(* 
:Description: This function block is base for all other measurement fixtures.
*)
FUNCTION_BLOCK ABSTRACT FB_UniversalFixture IMPLEMENTS  I_UniversalFixture
VAR CONSTANT
	sSAMPLE_ACCEPTED : STRING := 'ACCEPTED';					(* Sample accepted - compare keyword for TCP/IP message from measurement device *)
	sSAMPLE_REJECTED : STRING := 'REJECTED';					(* Sample rejected - compare keyword for TCP/IP message from measurement device *)
END_VAR
VAR
	bFirstCycle				: BOOL := TRUE;						(* First cycle bit *)
	sName 					: STRING; 							(* Fixture name for other utilities *)
	
	bActive 				: BOOL;								(* Fixture device is initialized and ready to wokr *)
	bBusy					: BOOL;								(* Fixture device is busy *)
	bError 					: BOOL;								(* Error occured while executing *)
	iErrorID 				: UDINT;							(* Error ID *)
	
	eSampleResult			: E_UniversalFixtureSampleResult;	(* Result of current measured product *)
	iSampleID				: UDINT;							(* Id of current measured product *)
	bSocketOpen				: BOOL;								(* Socket open flag *)
	
	sSendData				: STRING;							(* String message to send via TCP/IP to measurement device *)
	sRecivedData			: STRING;							(* String message to recive via TCP/IP from measurement device *)
	sLoggerMessage			: STRING;							(* String message for measurement txt logger *)
	stSendData				: ST_TcpBufferData;					(* Byte message to send via TCP/IP to measurement device *)
	stReciveData			: ST_TcpBufferData;					(* Byte message to recive via TCP/IP from measurement device *)
	fbTcpServer				: FB_TcpServer;						(* TCP/IP server instance *)
	fbTcpClient				: FB_TcpClient;						(* TCP/IP client instance *)
	bUseLogger				: BOOL;								(* Enables using of internal fixture file logger *)
	fbMeasurementLogger 	: FB_TXTDataExchanger;				(* Measurement TXT-File logger *)
	
	rtError					: R_TRIG; 							(* Rising edge trigger for function block error *)
	
	eFixtureState			: E_UniversalFixtureState;			(* Current state of measurement fixture device *)
	eFixtureStateInit		: E_UniversalFixtureStateInit;		(* Current state of measurement fixture device initialization *)
	eFixtureStateAbort		: E_UniversalFixtureStateAbort;		(* Current state of measurement fixture device aborting *)
	eFixtureStateReset		: E_UniversalFixtureStateReset;		(* Current state of measurement fixture device reseting *)
	eFixtureStateMeasure	: E_UniversalFixtureStateMeasure; 	(* Current measurement state if measurement has began *)
	eConnnectionType		: E_UniversalFixtureConnectionType;
	
	bClientConnection 		: BOOL; 							(* If true then fixture connect as a client, if false it behaves like a server *)
END_VAR

(* First cycle assignamnets *)
IF bFirstCycle THEN
	bFirstCycle := FALSE;
	
END_IF

(* Update status flags *)
bActive := eFixtureState >= UNIVERSAL_FIXTURE_READY;
bError := fbTcpServer.Error OR fbMeasurementLogger.Error;

(* Run server instance *)
IF eConnnectionType = UNIVERSAL_FIXTURE_SERVER_CONNECTION THEN
	fbTcpServer();
	
ELSIF eConnnectionType = UNIVERSAL_FIXTURE_CLIENT_CONNECTION THEN
	fbTcpClient();
	
END_IF 

(* Report errors that occur *)
rtError(CLK:=bError);

IF rtError.Q THEN 
	fbMachineLogger.MR_AddLogs(FUN_MergeStrings5(sName, ' : Error occured (error ID: ', UDINT_TO_STRING(iErrorID), ')', ''));
	
END_IF

(* Run internal measurement logger instance if it's enabled *)
IF bUseLogger THEN
	fbMeasurementLogger();
	
END_IF

(* Run main state machine *)
StateMachine();

PROPERTY Active : REFERENCE TO BOOL
GET
Active REF= bActive;
END_GET
END_PROPERTY

PROPERTY Busy : REFERENCE TO BOOL
GET
Busy REF= bBusy;
END_GET
END_PROPERTY

PROPERTY Error : REFERENCE TO BOOL
GET
Error REF= bError;
END_GET
END_PROPERTY

METHOD PROTECTED M_MeasurementClient : BOOL
VAR_INPUT
END_VAR
CASE eFixtureStateMeasure OF
	UNIVERSAL_FIXTURE_MEASURE_SEND_DATA:
		(* Prepare and send data to client *)
		sSendData := CONCAT('START;',UDINT_TO_STRING(iSampleID));
		sSendData := CONCAT(sSendData, '$R$N');
		FUN_StringToTcpBufferData(sMessageAddr := ADR(sSendData), stSendDataAddr := ADR(stSendData));
		fbTcpClient.MR_AppendToSendBuffer(stData := stSendData);
		
		(* Prepare data for logger *)
		IF bUseLogger THEN
			MEMSET(ADR(sLoggerMessage),0,INT_TO_UDINT(LEN(sLoggerMessage)));
			sLoggerMessage := CONCAT('SampleID:',UDINT_TO_STRING(iSampleID));
			
		END_IF
		
		eFixtureStateMeasure := UNIVERSAL_FIXTURE_MEASURE_RECIVE_DATA;
		
	UNIVERSAL_FIXTURE_MEASURE_RECIVE_DATA:
		stReciveData := fbTcpClient.NextRecivedMessage;
		
		IF stReciveData.iLength > 0 THEN
			FUN_TcpBufferDataToString(sMessageAddr := ADR(sRecivedData), stReturnDataAddr := ADR(stReciveData));
			
			(* Sample accepted *)
			IF MEMCMP(ADR(sRecivedData),ADR(sSAMPLE_ACCEPTED),INT_TO_UDINT(LEN(sSAMPLE_ACCEPTED))) = 0 THEN
				IF bUseLogger THEN
					sLoggerMessage := CONCAT(sLoggerMessage,sSAMPLE_ACCEPTED);
					fbMeasurementLogger.MR_AddLogs(sLoggerMessage);
					
				END_IF
				eSampleResult := UNIVERSAL_FIXTURE_SAMPLE_ACCEPTED;
				eFixtureStateMeasure := UNIVERSAL_FIXTURE_MEASURE_DONE;
				
			(* Sample rejected *)
			ELSIF MEMCMP(ADR(sRecivedData),ADR(sSAMPLE_REJECTED),INT_TO_UDINT(LEN(sSAMPLE_REJECTED))) = 0 THEN
				IF bUseLogger THEN
					sLoggerMessage := CONCAT(sLoggerMessage,sSAMPLE_REJECTED);
					fbMeasurementLogger.MR_AddLogs(sLoggerMessage);
					
				END_IF
				eSampleResult := UNIVERSAL_FIXTURE_SAMPLE_REJECTED;
				eFixtureStateMeasure := UNIVERSAL_FIXTURE_MEASURE_DONE;
				
			END_IF
		END_IF
		
	UNIVERSAL_FIXTURE_MEASURE_DONE:
		fbTcpClient.MR_ClearAllBuffers();
		eFixtureStateMeasure := UNIVERSAL_FIXTURE_MEASURE_SEND_DATA;
		eFixtureState := UNIVERSAL_FIXTURE_METHOD_DONE;
		
END_CASE
END_METHOD

METHOD PROTECTED M_MeasurementServer : BOOL
VAR_INPUT
END_VAR
CASE eFixtureStateMeasure OF
	UNIVERSAL_FIXTURE_MEASURE_WAIT_FOR_CLIENT:
		IF fbTcpServer.ServerState = TCPIP_SERVER_RUNNING_DATA_EXCHANGE THEN
			eFixtureStateMeasure := UNIVERSAL_FIXTURE_MEASURE_SEND_DATA;
		END_IF
		
	UNIVERSAL_FIXTURE_MEASURE_SEND_DATA:
		(* Prepare and send data to client *)
		sSendData := CONCAT('START;',UDINT_TO_STRING(iSampleID));
		sSendData := CONCAT(sSendData, '$R$N');
		FUN_StringToTcpBufferData(sMessageAddr := ADR(sSendData), stSendDataAddr := ADR(stSendData));
		fbTcpServer.MR_AppendToSendBuffer(stData := stSendData);
		
		(* Prepare data for logger *)
		IF bUseLogger THEN
			MEMSET(ADR(sLoggerMessage),0,INT_TO_UDINT(LEN(sLoggerMessage)));
			sLoggerMessage := CONCAT('SampleID:',UDINT_TO_STRING(iSampleID));
		END_IF
		
		eFixtureStateMeasure := UNIVERSAL_FIXTURE_MEASURE_RECIVE_DATA;
		
	UNIVERSAL_FIXTURE_MEASURE_RECIVE_DATA:
		stReciveData := fbTcpServer.LastRecivedMessage;
		IF stReciveData.iLength > 0 THEN
			FUN_TcpBufferDataToString(sMessageAddr := ADR(sRecivedData), stReturnDataAddr := ADR(stReciveData));
			
			(* Sample accepted *)
			IF MEMCMP(ADR(sRecivedData),ADR(sSAMPLE_ACCEPTED),INT_TO_UDINT(LEN(sSAMPLE_ACCEPTED))) = 0 THEN
				IF bUseLogger THEN
					sLoggerMessage := CONCAT(sLoggerMessage,sSAMPLE_ACCEPTED);
					fbMeasurementLogger.MR_AddLogs(sLoggerMessage);
				END_IF
				eSampleResult := UNIVERSAL_FIXTURE_SAMPLE_ACCEPTED;
				eFixtureStateMeasure := UNIVERSAL_FIXTURE_MEASURE_DONE;
				
			(* Sample rejected *)
			ELSIF MEMCMP(ADR(sRecivedData),ADR(sSAMPLE_REJECTED),INT_TO_UDINT(LEN(sSAMPLE_REJECTED))) = 0 THEN
				IF bUseLogger THEN
					sLoggerMessage := CONCAT(sLoggerMessage,sSAMPLE_REJECTED);
					fbMeasurementLogger.MR_AddLogs(sLoggerMessage);
				END_IF
				eSampleResult := UNIVERSAL_FIXTURE_SAMPLE_REJECTED;
				eFixtureStateMeasure := UNIVERSAL_FIXTURE_MEASURE_DONE;
				
			END_IF
		END_IF
		
	UNIVERSAL_FIXTURE_MEASURE_DONE:
		fbTcpServer.MR_ClearAllBuffers();
		eFixtureStateMeasure := UNIVERSAL_FIXTURE_MEASURE_WAIT_FOR_CLIENT;
		eFixtureState := UNIVERSAL_FIXTURE_METHOD_DONE;
		
END_CASE
END_METHOD

METHOD MR_Abort : BOOL
IF eFixtureState >= UNIVERSAL_FIXTURE_INITIALIZING THEN
	bBusy := TRUE;
	MR_Abort := FALSE;
	eFixtureState := UNIVERSAL_FIXTURE_ABORTING;
	fbMachineLogger.MR_AddLogs(CONCAT(sName,' : abort requested'));	

ELSIF eFixtureState = UNIVERSAL_FIXTURE_UNINITIALIZED THEN
	bBusy := FALSE;
	MR_Abort := TRUE;
	fbMachineLogger.MR_AddLogs(CONCAT(sName,' : abort done'));	

END_IF
END_METHOD

METHOD MR_Close : BOOL
IF eFixtureState = UNIVERSAL_FIXTURE_IDLE AND THIS^.SocketOpen THEN
	bBusy := TRUE;	
	MR_Close := FALSE;
	eFixtureState := UNIVERSAL_FIXTURE_CLOSE;
	fbMachineLogger.MR_AddLogs(CONCAT(sName,' : close requested'));	
	
ELSIF eFixtureState = UNIVERSAL_FIXTURE_METHOD_DONE THEN
	bBusy := FALSE;
	MR_Close := TRUE;
	fbMachineLogger.MR_AddLogs(CONCAT(sName,' : close done'));	

END_IF
END_METHOD

METHOD MR_FirstCycle : BOOL
VAR_INPUT
	sFixtureName 		: STRING;		(*  *)
	sHost				: T_IPv4Addr;	(*  *)
	sAmsNetID 			: T_AmsNetID;	(*  *)
	iPort				: UINT;			(*  *)
	tTimeout			: TIME;			(*  *)
	bUseLogger			: BOOL;			(*  *)
	bClientConnection 	: BOOL;			(*  *)
	sFileDir			: STRING;		(*  *)
	sFileName			: STRING;		(*  *)
	bCreateFileAtStart	: BOOL;
	bAddHeader			: BOOL;
	bAddTimeStamp		: BOOL;	
END_VAR
THIS^.sName := sFixtureName;
THIS^.bUseLogger := bUseLogger;
THIS^.bClientConnection := bClientConnection;

IF THIS^.bClientConnection THEN 
	(* Set fixture client initial parameters *)
	THIS^.fbTcpClient.MR_FirstCycle(	sName 		:= CONCAT('TCP/IP client of ',sFixtureName),
										sHost		:= sHost,
										sAmsNetID	:= sAmsNetID,
										iPort 		:= iPort,
										tTimeout 	:= tTimeout);	
ELSE
	(* Set fixture server initial parameters *)
	THIS^.fbTcpServer.MR_FirstCycle(	sName 		:= CONCAT('TCP/IP server of ',sFixtureName),
										sHost		:= sHost,
										sAmsNetID	:= sAmsNetID,
										iPort 		:= iPort,
										tTimeout 	:= tTimeout);
END_IF								
									
IF THIS^.bUseLogger THEN
	(* Set measurement logger initial parameters*)									
	THIS^.fbMeasurementLogger.MR_FirstCycle(sName 	:= sName,
											sFileDir 	:= sFileDir,
											sFileName 	:= sFileName,
											sAmsNetId 	:= '',
											bCreateFileAtStart := bCreateFileAtStart,
											bAddHeader 	:= bAddHeader,
											bAddTimeStamp := bAddTimeStamp);	
END_IF
END_METHOD

METHOD MR_Init : BOOL
IF eFixtureState = UNIVERSAL_FIXTURE_UNINITIALIZED THEN
	bBusy := TRUE;
	MR_Init := FALSE;
	
	IF bClientConnection THEN 
		eConnnectionType := UNIVERSAL_FIXTURE_CLIENT_CONNECTION;
		eFixtureStateInit := UNIVERSAL_FIXTURE_INIT_TCP_CLIENT;
		
	ELSE
		eConnnectionType := UNIVERSAL_FIXTURE_SERVER_CONNECTION;	
		eFixtureStateInit := UNIVERSAL_FIXTURE_INIT_TCP_SERVER;	
		
	END_IF
	
	eFixtureState := UNIVERSAL_FIXTURE_INITIALIZING;
	fbMachineLogger.MR_AddLogs(CONCAT(sName,' : initialization requested'));	
	
ELSIF eFixtureState >= UNIVERSAL_FIXTURE_READY THEN
	bBusy := FALSE;
	MR_Init := TRUE;
	fbMachineLogger.MR_AddLogs(CONCAT(sName,' : initialization done'));
	
END_IF
END_METHOD

METHOD MR_Measure : BOOL
VAR_INPUT
	iSampleID : UINT;
END_VAR
IF eFixtureState = UNIVERSAL_FIXTURE_IDLE THEN
	bBusy := TRUE;
	MR_Measure := FALSE;
	THIS^.iSampleID := iSampleID;
	THIS^.eSampleResult := UNIVERSAL_FIXTURE_SAMPLE_UNKNOWN;
	
	IF eConnnectionType = UNIVERSAL_FIXTURE_SERVER_CONNECTION THEN
		eFixtureStateMeasure := UNIVERSAL_FIXTURE_MEASURE_WAIT_FOR_CLIENT;
		
	ELSIF eConnnectionType = UNIVERSAL_FIXTURE_CLIENT_CONNECTION THEN
		eFixtureStateMeasure := UNIVERSAL_FIXTURE_MEASURE_SEND_DATA;
		
	END_IF
	
	eFixtureState := UNIVERSAL_FIXTURE_MEASUREMENT;
	fbMachineLogger.MR_AddLogs(CONCAT(sName,' : measurement requested'));	

ELSIF eFixtureState = UNIVERSAL_FIXTURE_METHOD_DONE THEN
	bBusy := FALSE;
	MR_Measure := TRUE;
	fbMachineLogger.MR_AddLogs(CONCAT(sName,' : measurement done'));	
	
END_IF
END_METHOD

METHOD MR_Open : BOOL
IF eFixtureState = UNIVERSAL_FIXTURE_IDLE AND NOT THIS^.SocketOpen THEN
	bBusy := TRUE;
	MR_Open := FALSE;
	eFixtureState := UNIVERSAL_FIXTURE_OPEN;
	fbMachineLogger.MR_AddLogs(CONCAT(sName,' : open requested'));		
	
ELSIF eFixtureState = UNIVERSAL_FIXTURE_METHOD_DONE THEN
	bBusy := FALSE;
	MR_Open := TRUE;
	fbMachineLogger.MR_AddLogs(CONCAT(sName,' : open done'));		
	
END_IF
END_METHOD

METHOD MR_Reset : BOOL
IF eFixtureState >= UNIVERSAL_FIXTURE_IDLE AND bError THEN
	bBusy := TRUE;
	MR_Reset := FALSE;
	eFixtureState := UNIVERSAL_FIXTURE_RESET;
	fbMachineLogger.MR_AddLogs(CONCAT(sName,' : reset requested'));			
	
ELSIF eFixtureState = UNIVERSAL_FIXTURE_METHOD_DONE THEN
	bBusy := FALSE;
	MR_Reset := TRUE;
	fbMachineLogger.MR_AddLogs(CONCAT(sName,' : reset done'));			
	
END_IF
END_METHOD

METHOD PROTECTED MS_Aborting
VAR_INPUT
END_VAR
CASE eFixtureStateAbort OF
	UNIVERSAL_FIXTURE_ABORT_FILE_LOGGER:
		IF bUseLogger THEN
			fbMeasurementLogger.MR_Abort();
		
			IF NOT fbMeasurementLogger.Busy THEN
				IF eConnnectionType = UNIVERSAL_FIXTURE_SERVER_CONNECTION THEN
					eFixtureStateAbort := UNIVERSAL_FIXTURE_ABORT_TCP_SERVER;
					
				ELSIF eConnnectionType = UNIVERSAL_FIXTURE_CLIENT_CONNECTION THEN
					eFixtureStateAbort := UNIVERSAL_FIXTURE_ABORT_TCP_CLIENT;
					
				END_IF
			END_IF
		ELSE
			IF eConnnectionType = UNIVERSAL_FIXTURE_SERVER_CONNECTION THEN
				eFixtureStateAbort := UNIVERSAL_FIXTURE_ABORT_TCP_SERVER;
				
			ELSIF eConnnectionType = UNIVERSAL_FIXTURE_CLIENT_CONNECTION THEN
				eFixtureStateAbort := UNIVERSAL_FIXTURE_ABORT_TCP_CLIENT;
				
			END_IF
		END_IF
		
	UNIVERSAL_FIXTURE_ABORT_TCP_SERVER:
		fbTcpServer.MR_Abort();
		
		IF NOT fbTcpServer.Active THEN
			eFixtureStateAbort := UNIVERSAL_FIXTURE_ABORT_DONE;
			
		END_IF

	UNIVERSAL_FIXTURE_ABORT_TCP_CLIENT:
		fbTcpClient.MR_Abort();
		
		IF NOT fbTcpClient.Active THEN
			eFixtureStateAbort := UNIVERSAL_FIXTURE_ABORT_DONE;
			
		END_IF
		
	UNIVERSAL_FIXTURE_ABORT_DONE:
		eFixtureStateAbort := UNIVERSAL_FIXTURE_ABORT_FILE_LOGGER;
		eFixtureState := UNIVERSAL_FIXTURE_UNINITIALIZED;
	
END_CASE
END_METHOD

METHOD PROTECTED ABSTRACT MS_Close
VAR_INPUT
END_VAR
;
END_METHOD

METHOD PROTECTED MS_Extension
VAR_INPUT
END_VAR
END_METHOD

METHOD PROTECTED MS_Idle
VAR_INPUT
END_VAR
;
END_METHOD

METHOD PROTECTED MS_Initializing
VAR_INPUT
END_VAR
CASE eFixtureStateInit OF
	UNIVERSAL_FIXTURE_INIT_TCP_SERVER:
		fbTcpServer.MR_Init();
		
		IF fbTcpServer.Active THEN
			eFixtureStateInit := UNIVERSAL_FIXTURE_INIT_FILE_LOGGER;
			
		END_IF

	UNIVERSAL_FIXTURE_INIT_TCP_CLIENT:
		fbTcpClient.MR_Init();
		
		IF fbTcpClient.Active THEN
			eFixtureStateInit := UNIVERSAL_FIXTURE_INIT_FILE_LOGGER;
			
		END_IF
		
	UNIVERSAL_FIXTURE_INIT_FILE_LOGGER:
		IF bUseLogger THEN
			fbMeasurementLogger.MR_Init();
		
			IF fbMeasurementLogger.Busy THEN
				eFixtureStateInit := UNIVERSAL_FIXTURE_INIT_DONE;
				
			END_IF
		ELSE
			eFixtureStateInit := UNIVERSAL_FIXTURE_INIT_DONE;
			
		END_IF
		
	UNIVERSAL_FIXTURE_INIT_DONE:
		eFixtureStateInit := UNIVERSAL_FIXTURE_INIT_TCP_SERVER;
		eFixtureState := UNIVERSAL_FIXTURE_READY;
	
END_CASE
END_METHOD

METHOD PROTECTED MS_Measurement
VAR_INPUT
END_VAR
IF eConnnectionType = UNIVERSAL_FIXTURE_SERVER_CONNECTION THEN
	M_MeasurementServer();
	
ELSIF eConnnectionType = UNIVERSAL_FIXTURE_CLIENT_CONNECTION THEN
	M_MeasurementClient();
	
END_IF
END_METHOD

METHOD PROTECTED MS_MethodDone
VAR_INPUT
END_VAR
IF NOT bBusy THEN
	eFixtureState := UNIVERSAL_FIXTURE_IDLE;
	
END_IF
END_METHOD

METHOD PROTECTED ABSTRACT MS_Open
VAR_INPUT
END_VAR
END_METHOD

METHOD PROTECTED MS_Ready
VAR_INPUT
END_VAR
eFixtureState := UNIVERSAL_FIXTURE_IDLE;
END_METHOD

METHOD PROTECTED MS_Reset
VAR_INPUT
END_VAR
CASE eFixtureStateReset OF 
	UNIVERSAL_FIXTURE_RESETING_FILE_LOGGER:
		IF bUseLogger THEN
			fbMeasurementLogger.MR_Reset();
		
			IF NOT fbMeasurementLogger.Busy THEN
				IF eConnnectionType = UNIVERSAL_FIXTURE_SERVER_CONNECTION THEN
					eFixtureStateReset := UNIVERSAL_FIXTURE_RESETING_TCP_SERVER_SHUT_DOWN;
					
				ELSIF eConnnectionType = UNIVERSAL_FIXTURE_CLIENT_CONNECTION THEN
					eFixtureStateReset := UNIVERSAL_FIXTURE_RESETING_TCP_CLIENT_SHUT_DOWN;
					
				END_IF
			END_IF
		ELSE
			IF eConnnectionType = UNIVERSAL_FIXTURE_SERVER_CONNECTION THEN
				eFixtureStateReset := UNIVERSAL_FIXTURE_RESETING_TCP_SERVER_SHUT_DOWN;
				
			ELSIF eConnnectionType = UNIVERSAL_FIXTURE_CLIENT_CONNECTION THEN
				eFixtureStateReset := UNIVERSAL_FIXTURE_RESETING_TCP_CLIENT_SHUT_DOWN;
				
			END_IF
		END_IF
		
	UNIVERSAL_FIXTURE_RESETING_TCP_SERVER_SHUT_DOWN:
		fbTcpServer.MR_Abort();
		
		IF NOT fbTcpServer.Active THEN
			eFixtureStateReset := UNIVERSAL_FIXTURE_RESETING_TCP_SERVER_TURN_ON;
			
		END_IF
		
	UNIVERSAL_FIXTURE_RESETING_TCP_SERVER_TURN_ON:
		fbTcpServer.MR_Init();
		
		IF fbTcpServer.Active THEN
			eFixtureStateReset := UNIVERSAL_FIXTURE_RESETING_DONE;
			
		END_IF

	UNIVERSAL_FIXTURE_RESETING_TCP_CLIENT_SHUT_DOWN:
		fbTcpClient.MR_Abort();
		
		IF NOT fbTcpClient.Active THEN
			eFixtureStateReset := UNIVERSAL_FIXTURE_RESETING_TCP_CLIENT_TURN_ON;
			
		END_IF
		
	UNIVERSAL_FIXTURE_RESETING_TCP_CLIENT_TURN_ON:
		fbTcpClient.MR_Init();
		
		IF fbTcpClient.Active THEN
			eFixtureStateReset := UNIVERSAL_FIXTURE_RESETING_DONE;
			
		END_IF
		
	UNIVERSAL_FIXTURE_RESETING_DONE:		
		bError := FALSE;
		
		eFixtureStateReset := UNIVERSAL_FIXTURE_RESETING_FILE_LOGGER;
		eFixtureState := UNIVERSAL_FIXTURE_METHOD_DONE;
		
END_CASE
END_METHOD

METHOD PROTECTED MS_Uninitialized
VAR_INPUT
END_VAR
bBusy := FALSE;
bError := FALSE;
iErrorID := 0;
iSampleID := 0;

eSampleResult := UNIVERSAL_FIXTURE_SAMPLE_UNKNOWN;
END_METHOD

PROPERTY RecivedUtuData : REFERENCE TO STRING
GET
RecivedUtuData REF= sRecivedData;
END_GET
END_PROPERTY

PROPERTY ref_MeasurementLogger : REFERENCE TO FB_TXTDataExchanger
GET
ref_MeasurementLogger REF= fbMeasurementLogger;
END_GET
END_PROPERTY

PROPERTY ref_TcpClient : REFERENCE TO FB_TcpClient
GET
ref_TcpClient REF= fbTcpClient;
END_GET
END_PROPERTY

PROPERTY ref_TcpServer : REFERENCE TO FB_TcpServer
GET
ref_TcpServer REF= fbTcpServer;
END_GET
END_PROPERTY

PROPERTY SampleID : REFERENCE TO UDINT
GET
SampleID REF= iSampleID;
END_GET
END_PROPERTY

PROPERTY SampleResult : REFERENCE TO E_UniversalFixtureSampleResult
GET
SampleResult REF= eSampleResult;
END_GET
END_PROPERTY

PROPERTY ABSTRACT SocketOpen : REFERENCE TO BOOL
GET
END_GET
END_PROPERTY

PROPERTY State : REFERENCE TO E_UniversalFixtureState
GET
State REF= eFixtureState;
END_GET
END_PROPERTY

METHOD PROTECTED StateMachine
VAR_INPUT
END_VAR
CASE eFixtureState OF
	UNIVERSAL_FIXTURE_UNINITIALIZED:
		MS_Uninitialized();
		
	UNIVERSAL_FIXTURE_INITIALIZING:
		MS_Initializing();
		
	UNIVERSAL_FIXTURE_READY:
		MS_Ready();
		
	UNIVERSAL_FIXTURE_IDLE:
		MS_Idle();
	
	UNIVERSAL_FIXTURE_OPEN:
		MS_Open();
		
	UNIVERSAL_FIXTURE_CLOSE:
		MS_Close();
	
	UNIVERSAL_FIXTURE_MEASUREMENT:
		MS_Measurement();
	
	UNIVERSAL_FIXTURE_RESET:
		MS_Reset();
		
	UNIVERSAL_FIXTURE_METHOD_DONE:
		MS_MethodDone();
		
	UNIVERSAL_FIXTURE_EXTENSION:
		MS_Extension();
	
	UNIVERSAL_FIXTURE_ABORTING:
		MS_Aborting();
	
END_CASE
END_METHOD

END_FUNCTION_BLOCK

(* stored: Version 1.1.0.1, ProductVersion 3.1.4024.9
   POU FB_UniversalFixture: Id {871ce81f-e673-4772-aced-b3c5dd104678}, SpecialFunc None
   Folder FirstCycle: Id {6ac848c3-8849-420d-9545-ab512f6fc4bd}
   Folder Internal: Id {ee5fedc1-8906-4cf6-8983-a137bf6000f4}
   Folder Properties: Id {2a131754-db76-4f9b-8a4e-4f30746c4409}
   Folder References: Id {45360bee-050b-4e56-aee3-4609f5cce1d5}
   Folder Status: Id {db161780-2258-42e8-9377-940a048dd600}
   Folder Requests: Id {26310939-11e6-4da6-a46c-7469a248a566}
   Folder StateMachine: Id {c657b9b2-0d96-4635-bfd8-c36ce219a6e0}
   Property Active: Id {1cc65cf1-7e33-42d6-83d6-557ea8985d18}
   Get Get: Id {f16a351b-a11c-46e5-99e0-ae9c6d0b1588}
   Property Busy: Id {9930e1cd-28f5-4631-b6e2-6732b10b85bd}
   Get Get: Id {2ed76f81-35b8-496c-b07e-a25e46ec6514}
   Property Error: Id {473cc5f2-97bd-40ed-a7b6-76a06c7d6131}
   Get Get: Id {26531b75-ecec-4e06-8005-46266d0429cd}
   Method M_MeasurementClient: Id {88cb3cca-71f4-425d-9c2b-45da1987ac06}
   Method M_MeasurementServer: Id {09f740ba-5846-4b85-bcc9-58f44a7c5edd}
   Method MR_Abort: Id {5f8a8145-8308-450c-80b3-bea419e7a94d}
   Method MR_Close: Id {bcd26b28-6c76-4c74-8e76-db1e0c1c5310}
   Method MR_FirstCycle: Id {47401250-f48c-4724-9c74-af31e541cf35}
   Method MR_Init: Id {7c351ee9-672b-4dd3-b865-53ec6bf38c04}
   Method MR_Measure: Id {ac3d07ac-d5c3-42b3-9992-7300d79437ca}
   Method MR_Open: Id {604d37b9-b7ce-4ab0-94e2-2b3fe3f12c2a}
   Method MR_Reset: Id {55354bfc-3c36-4a98-b13c-5b9230f8ad97}
   Method MS_Aborting: Id {c38cff8a-e0b9-4473-b0c9-97e41f0daae4}
   Method MS_Close: Id {a819e8dd-884b-4d3f-9df3-835929036c45}
   Method MS_Extension: Id {903d0d4f-1bfe-4c3e-acbc-58e4d09cdf8d}
   Method MS_Idle: Id {85566248-c2a8-4e79-99c4-2e8fe8a8a873}
   Method MS_Initializing: Id {a90277bb-d087-43a9-ba52-2ff6745bcac2}
   Method MS_Measurement: Id {fb3bcf01-367f-4b90-9de9-fd0e26fc8ef2}
   Method MS_MethodDone: Id {b0647aad-660b-4949-a3f6-1cf0162fdcc2}
   Method MS_Open: Id {3f120c87-457b-4875-8ad5-734001404a75}
   Method MS_Ready: Id {69c5e074-7e01-4447-a764-ed1f3d3ab3ee}
   Method MS_Reset: Id {bd357273-8fe0-4806-a7e3-4fc0e5007688}
   Method MS_Uninitialized: Id {b9924a38-15e9-44b5-9438-f5e4ad2f8911}
   Property RecivedUtuData: Id {d2625672-f7a5-46ef-b253-fa6f9f7e9b01}
   Get Get: Id {92b85f34-b721-4575-86a3-6017bffeae49}
   Property ref_MeasurementLogger: Id {63ca4ed3-2edd-4b48-992b-89b0d334d147}
   Get Get: Id {eaf5792e-5228-44d2-9c06-90e147c3796d}
   Property ref_TcpClient: Id {3d5c1726-81d4-4d46-bad0-37dcf914ec41}
   Get Get: Id {3c0fb401-f63d-4ee9-89d5-499c868c714c}
   Property ref_TcpServer: Id {478b11d8-32dd-4213-acb6-849aeba91fbe}
   Get Get: Id {d4ac500e-8421-4aee-bd4d-073205767940}
   Property SampleID: Id {0ede5fc3-f149-44c3-9a53-8c5142068224}
   Get Get: Id {ca142f3e-13db-408a-bd82-862f6745fd7d}
   Property SampleResult: Id {9ad07b45-f2b4-4ec1-afdb-e91d00e44189}
   Get Get: Id {c968e653-0bd4-4e1e-86fe-2d1ca8ac8ac0}
   Property SocketOpen: Id {9e548cf6-2ea3-47cf-ae0d-a35532f263a1}
   Get Get: Id {e663fbeb-cb4a-40bb-97b9-c70af3da3e95}
   Property State: Id {ae000683-58a7-4d3e-93ab-0d2ff59bbf18}
   Get Get: Id {40e2329a-65ee-453c-8d33-841d0fcf28fd}
   Method StateMachine: Id {5ac9923d-cd36-48db-8851-002b5c67d068} *)
